(* IEC 61131-3 sources: RL_MAR/experiments/comparison/autoplc/results/gpt-4o-mini_20260511_164212/med_81, 1 file *)

(* ---- med_81_1.st ---- *)
FUNCTION_BLOCK SolarPanelTracking
VAR
    PanelAngle : REAL; (* Output for adjusting the solar panel angle *)
    SunriseTime : TIME := T#6H; (* Set the time for sunrise (6:00 AM) *)
    SunsetTime : TIME := T#18H; (* Set the time for sunset (6:00 PM) *)
    NoonTime : TIME := T#12H; (* Set the time for solar noon (12:00 PM) *)
    MorningAngle : REAL := 30.0; (* Set the morning angle for panels *)
    NoonAngle : REAL := 60.0; (* Set the noon angle for panels *)
    EveningAngle : REAL := 30.0; (* Set the evening angle for panels *)
END_VAR

VAR_INPUT
    CurrentTime : TIME; (* Current time input from the PLC's real-time clock *)
    SolarIntensity : REAL; (* Measured solar intensity input *)
END_VAR

(* Control Logic Implementation *)
IF SolarIntensity >= 90.0 THEN
    PanelAngle := NoonAngle; (* Override to NoonAngle if solar intensity is high *)
ELSE
    IF (CurrentTime < SunriseTime) OR (CurrentTime >= SunsetTime) THEN
        PanelAngle := 0.0; (* Nighttime: set to horizontal *)
    ELSIF (CurrentTime >= SunriseTime) AND (CurrentTime < NoonTime) THEN
        PanelAngle := MorningAngle; (* Morning: set to morning angle *)
    ELSIF (CurrentTime >= NoonTime) AND (CurrentTime < SunsetTime) THEN
        PanelAngle := EveningAngle; (* Afternoon/Evening: set to evening angle *)
    END_IF;
END_IF;

END_FUNCTION_BLOCK
